(* PLC project Generated.project, CODESYS CODESYS V3.5 SP19 Patch 1 *)
(* stored: creationDateTime 2026-09-01T00:57:57.885332, modificationDateTime 2026-09-01T00:57:57.885332 *)

(* ═══════════════════════════════════════════════════════════════ 🪨 ST_CycleDumpAtTremieHMI — Échange IHM cycle vidage trémie (legacy) ═══════════════════════════════════════════════════════════════ *)
TYPE ST_CycleDumpAtTremieHMI : STRUCT
  Cmd : ST_CycleDumpAtTremieCmd;
  State : ST_CycleDumpAtTremieState;
  Cfg : ST_CycleDumpAtTremieCfg;
END_STRUCT;
END_TYPE

(* ═══════════════════════════════════════════════════════════════ ⚙️ ST_CycleDumpAtTremieCfg — Réglages persistants cycle vidage trémie (legacy) ═══════════════════════════════════════════════════════════════ *)
TYPE ST_CycleDumpAtTremieCfg : STRUCT
  Initialized : BOOL := FALSE;  (* 🚦 flag restauration boot *)
END_STRUCT;
END_TYPE

(* ═══════════════════════════════════════════════════════════════ 🎮 ST_CycleDumpAtTremieCmd — Sélections IHM cycle vidage trémie (legacy) ═══════════════════════════════════════════════════════════════ *)
TYPE ST_CycleDumpAtTremieCmd : STRUCT
  TglEnableDumpAtTremie : BOOL := FALSE;  (* Mode vidage à la trémie — RESTREINT des mouvements dès le boot *)
END_STRUCT;
END_TYPE

(* ═══════════════════════════════════════════════════════════════ 🚦 ST_CycleDumpAtTremieState — États publics cycle vidage trémie (legacy) ═══════════════════════════════════════════════════════════════ *)
TYPE ST_CycleDumpAtTremieState : STRUCT
  DumpAtTremieArmed : BOOL;  (* TglEnableDumpAtTremie (bit IHM brut) *)
  DumpAtTremieAssistActive : BOOL;  (* Armé ET Mode MAINT_N1/N2 (mode réellement actif) *)
  DumpAtTremieAtTremie : BOOL;  (* M3_AtTremieStable *)
  DumpAtTremieBucketOpenArmed : BOOL;  (* CmdOpen_IHM déclenché par ce mode *)
  DumpAtTremieDescentLocked : BOOL;  (* DescendPermit M1/M2 forcé par ce mode (hors P1/Maintenance) *)
END_STRUCT;
END_TYPE
